INTERFACE IPAFMixing EXTENDS IPAProcessFunction

END_INTERFACE

(* stored: Version 1.1.0.1, ProductVersion 3.1.4020.12
   Itf IPAFMixing: Id {c1628cb2-5cc0-4224-a26a-8fc2fd25b8ae} *)
